TYPE ST_ChangeAllocate :
STRUCT
		Info 						: ST_NeedleChangeAllocateInfo;
		Handshake					: ST_HandshakeBase;
END_STRUCT
END_TYPE

(* stored: Version 1.1.0.1, ProductVersion 3.1.4024.13
   DUT ST_ChangeAllocate: Id {fc1f884f-e53b-4278-931e-6bde4f5bc18b} *)
